(* Schneider Machine Expert - Basic project correto_CORRIGIDO, file version 2.9.0.0 *)
(* ProjectInformations: Name=Novo projeto *)

HARDWARE
  Cpu 0: TM200CE24R
  ModuleExtensionObject 0: TM3TI4/G
  EthernetConfiguration: NetworkName=M200, IpAllocationMode=FixedAddress, IpAddress=192.168.10.1, SubnetMask=255.255.255.0
  SerialLineConfiguration: Baud=Baud9600, Parity=ParityNone, DataBits=DataBits8, StopBits=StopBits1, PhysicalMedium=PhysicalMediumRs485, TransmissionMode=TransmissionModeModbusRtu, SlaveId=1, Addressing=SlaveAddressing
  MastTask: UsePeriodScanMode=true, PeriodScan=10
  FastTask: Period=255
  CpuBehavior: StartingMode=StartAsPreviousState, AutoSaveRamOnEeprom=true, WatchdogPeriod=250

SYMBOLS  (address, symbol, comment, settings)
  %M100     MEM_I00
  %M101     MEM_I01
  %M102     MEM_I02
  %M103     MEM_I03
  %M104     MEM_I04
  %M105     MEM_I05
  %M106     MEM_I06
  %M107     MEM_I07
  %M108     MEM_I08
  %TM0        [Preset=6]
  %TM1        [Preset=2, Base=OneSecond]
  %I0.0     DJ_GERAL_ABERTO
  %I0.1     DJ_GERAL_FECHADO
  %I0.2     RESERVA1
  %I0.3     RESERVA2
  %I0.4     RESERVA3
  %I0.5     RESERVA4
  %I0.6     RESERVA5
  %I0.7     RESERVA6
  %I0.8     RESERVA7
  %I0.9     RESERVA8
  %I0.10    STS_SERVICO_AUX
  %I0.11    BOTAO_CLOSE
  %I0.12    BOTAO_OPEN
  %I0.13    BOTAO_EMERGENCIA
  %Q0.0     COMM_OK
  %Q0.1     USINAGERANDO
  %Q0.2     FALHA
  %Q0.3     ALARME
  %Q0.4     EMERGENCIA_INV
  %Q0.5     RESET_RASP
  %Q0.6     RESET_LINK_3G
  %Q0.7     RESERVA_1
  %Q0.8     RESERVA_2
  %Q0.9     RESERVA_3
  %IW1.0    TEMP_AMBIENTE  [Type=Type_PT100, Scope=Scope_Celsius, Minimum=-2000, Maximum=8500]
  %IW1.1    TEMP_QUADRO  [Type=Type_PT100, Scope=Scope_Celsius, Minimum=-2000, Maximum=8500]
  %IW1.2    TEMP_MODULO  [Type=Type_PT100, Scope=Scope_Celsius, Minimum=-2000, Maximum=8500]
  %IW1.3    TEMP_TRAFO  [Type=Type_PT100, Scope=Scope_Celsius, Minimum=-2000, Maximum=8500]

POU Saídas
  (* SectionNumber=1 *)

// Rung 0: COMUNICAÇÃO OK
  LD %M0
  ST %Q0.0                (* COMM_OK *)
  [ %MW600 := 1 ]
  // as ST:
  //   COMM_OK := %M0;
  //   IF %M0 THEN %MW600 := 1; END_IF;

// Rung 1: STATUS USINA GERANDO
  LD %M1
  ST %Q0.1                (* USINAGERANDO *)
  [ %MW601 := 1 ]
  // as ST:
  //   USINAGERANDO := %M1;
  //   IF %M1 THEN %MW601 := 1; END_IF;

// Rung 2: FALHA
  LD %M2
  ST %Q0.2                (* FALHA *)
  [ %MW602 := 1 ]
  // as ST:
  //   FALHA := %M2;
  //   IF %M2 THEN %MW602 := 1; END_IF;

// Rung 3: ALARME SONORO
  LD %M3
  ST %Q0.3                (* ALARME *)
  [ %MW603 := 1 ]
  // as ST:
  //   ALARME := %M3;
  //   IF %M3 THEN %MW603 := 1; END_IF;

// Rung 4: EMERGÊNCIA INVERSORES
  LDN %I0.13              (* BOTAO_EMERGENCIA *)
  OR %M4
  ST %Q0.4                (* EMERGENCIA_INV *)
  [ %MW604 := 1 ]
  // as ST:
  //   EMERGENCIA_INV := NOT BOTAO_EMERGENCIA OR %M4;
  //   IF NOT BOTAO_EMERGENCIA OR %M4 THEN %MW604 := 1; END_IF;

// Rung 5: RESET LINK 3G
  LD %M6
  ST %Q0.6                (* RESET_LINK_3G *)
  [ %MW606 := 1 ]
  // as ST:
  //   RESET_LINK_3G := %M6;
  //   IF %M6 THEN %MW606 := 1; END_IF;

// Rung 6: RESERVA
  LD %M7
  ST %Q0.7                (* RESERVA_1 *)
  // as ST:
  //   RESERVA_1 := %M7;

// Rung 7: RESERVA
  LD %M8
  ST %Q0.8                (* RESERVA_2 *)
  // as ST:
  //   RESERVA_2 := %M8;

// Rung 8: RESERVA
  LD %M9
  ST %Q0.9                (* RESERVA_3 *)
  // as ST:
  //   RESERVA_3 := %M9;

POU Entradas
  (* SectionNumber=2 *)

// Rung 9: STATUS DISJUNTOR GERAL ABERTO
  LD %I0.0                (* DJ_GERAL_ABERTO *)
  ST %M100                (* MEM_I00 *)
  [ %MW500 := 1 ]
  // as ST:
  //   MEM_I00 := DJ_GERAL_ABERTO;
  //   IF DJ_GERAL_ABERTO THEN %MW500 := 1; END_IF;

// Rung 10: STATUS DISJUNTOR GERAL FECHADO
  LD %I0.1                (* DJ_GERAL_FECHADO *)
  ST %M101                (* MEM_I01 *)
  [ %MW501 := 1 ]
  // as ST:
  //   MEM_I01 := DJ_GERAL_FECHADO;
  //   IF DJ_GERAL_FECHADO THEN %MW501 := 1; END_IF;

// Rung 11: RESERVA
  LD %I0.2                (* RESERVA1 *)
  ST %M102                (* MEM_I02 *)
  // as ST:
  //   MEM_I02 := RESERVA1;

// Rung 12: RESERVA
  LD %I0.3                (* RESERVA2 *)
  ST %M103                (* MEM_I03 *)
  // as ST:
  //   MEM_I03 := RESERVA2;

// Rung 13: RESERVA
  LD %I0.4                (* RESERVA3 *)
  ST %M104                (* MEM_I04 *)
  // as ST:
  //   MEM_I04 := RESERVA3;

// Rung 14: RESERVA
  LD %I0.5                (* RESERVA4 *)
  ST %M105                (* MEM_I05 *)
  // as ST:
  //   MEM_I05 := RESERVA4;

// Rung 15: RESERVA
  LD %I0.6                (* RESERVA5 *)
  ST %M106                (* MEM_I06 *)
  // as ST:
  //   MEM_I06 := RESERVA5;

// Rung 16: RESERVA
  LD %I0.7                (* RESERVA6 *)
  ST %M107                (* MEM_I07 *)
  // as ST:
  //   MEM_I07 := RESERVA6;

// Rung 17: RESERVA
  LD %I0.8                (* RESERVA7 *)
  ST %M108                (* MEM_I08 *)
  // as ST:
  //   MEM_I08 := RESERVA7;

// Rung 18: RESERVA
  LD %I0.9                (* RESERVA8 *)
  ST %M109
  // as ST:
  //   %M109 := RESERVA8;

// Rung 19: STATUS SERVIÇO AUXILIAR
  LD %I0.10               (* STS_SERVICO_AUX *)
  ST %M110
  [ %MW510 := 1 ]
  // as ST:
  //   %M110 := STS_SERVICO_AUX;
  //   IF STS_SERVICO_AUX THEN %MW510 := 1; END_IF;

// Rung 20: BOTÃO FECHA
  LD %I0.11               (* BOTAO_CLOSE *)
  ST %M111
  [ %MW511 := 1 ]
  // as ST:
  //   %M111 := BOTAO_CLOSE;
  //   IF BOTAO_CLOSE THEN %MW511 := 1; END_IF;

// Rung 21: BOTÃO ABRE
  LD %I0.12               (* BOTAO_OPEN *)
  ST %M112
  [ %MW512 := 1 ]
  // as ST:
  //   %M112 := BOTAO_OPEN;
  //   IF BOTAO_OPEN THEN %MW512 := 1; END_IF;

// Rung 22: BOTÃO EMERGÊNCIA
  LDN %I0.13              (* BOTAO_EMERGENCIA *)
  ST %M113
  [ %MW513 := 1 ]
  // as ST:
  //   %M113 := NOT BOTAO_EMERGENCIA;
  //   IF NOT BOTAO_EMERGENCIA THEN %MW513 := 1; END_IF;

POU Analógicas
  (* SectionNumber=3 *)

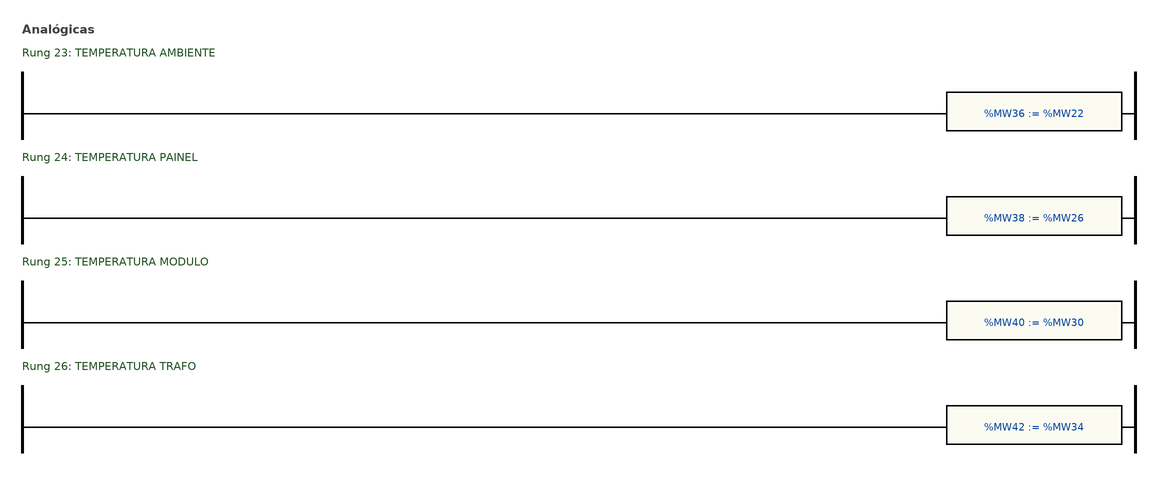

// Rung 23: TEMPERATURA AMBIENTE
  LD 1
  [ %MW36 := %MW22 ]
  // as ST:
  //   %MW36 := %MW22;

// Rung 24: TEMPERATURA PAINEL
  LD 1
  [ %MW38 := %MW26 ]
  // as ST:
  //   %MW38 := %MW26;

// Rung 25: TEMPERATURA MODULO
  LD 1
  [ %MW40 := %MW30 ]
  // as ST:
  //   %MW40 := %MW30;

// Rung 26: TEMPERATURA TRAFO
  LD 1
  [ %MW42 := %MW34 ]
  // as ST:
  //   %MW42 := %MW34;

POU ESCALA TEMPERATURA
  (* SectionNumber=4 *)

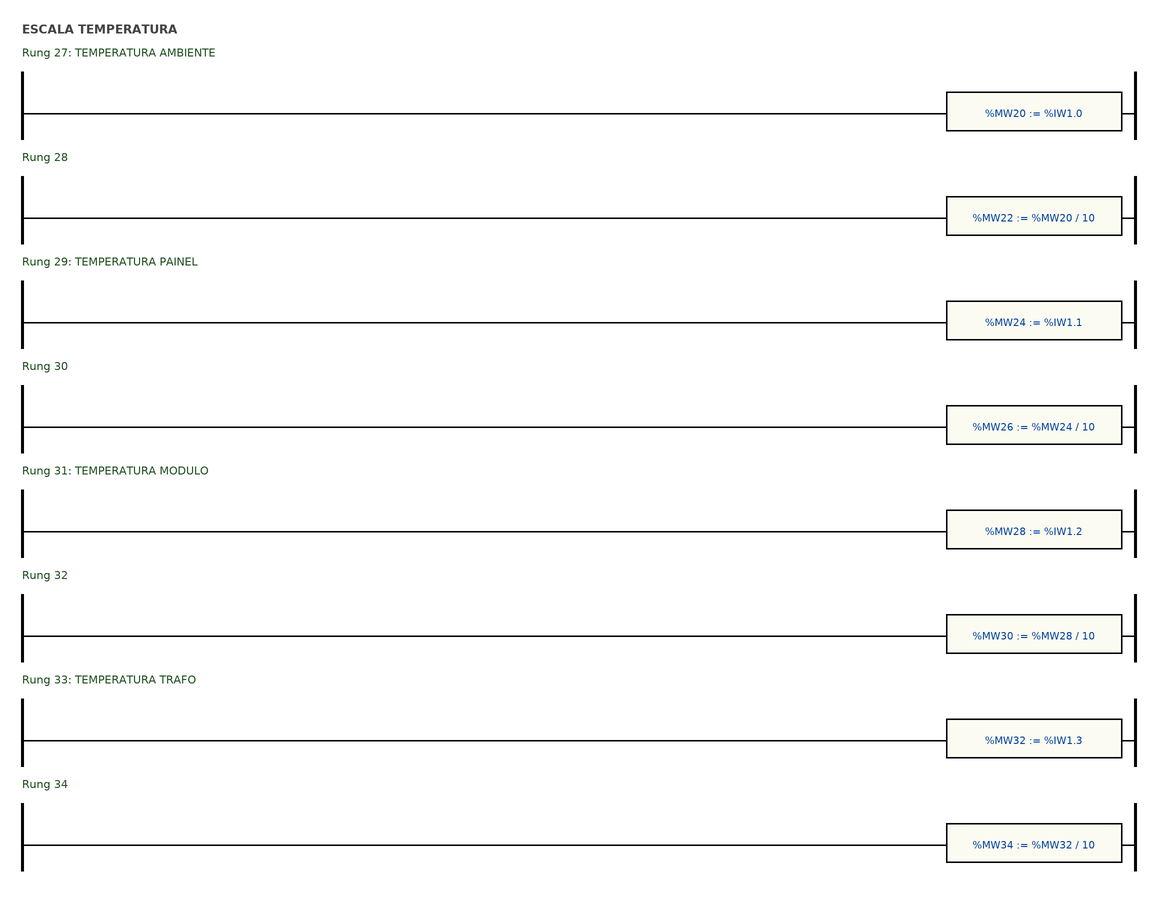

// Rung 27: TEMPERATURA AMBIENTE
  LD 1
  [ %MW20 := %IW1.0 ]     (* TEMP_AMBIENTE *)
  // as ST:
  //   %MW20 := TEMP_AMBIENTE;

// Rung 28
  LD 1
  [ %MW22 := %MW20 / 10 ]
  // as ST:
  //   %MW22 := %MW20 / 10;

// Rung 29: TEMPERATURA PAINEL
  LD 1
  [ %MW24 := %IW1.1 ]     (* TEMP_QUADRO *)
  // as ST:
  //   %MW24 := TEMP_QUADRO;

// Rung 30
  LD 1
  [ %MW26 := %MW24 / 10 ]
  // as ST:
  //   %MW26 := %MW24 / 10;

// Rung 31: TEMPERATURA MODULO
  LD 1
  [ %MW28 := %IW1.2 ]     (* TEMP_MODULO *)
  // as ST:
  //   %MW28 := TEMP_MODULO;

// Rung 32
  LD 1
  [ %MW30 := %MW28 / 10 ]
  // as ST:
  //   %MW30 := %MW28 / 10;

// Rung 33: TEMPERATURA TRAFO
  LD 1
  [ %MW32 := %IW1.3 ]     (* TEMP_TRAFO *)
  // as ST:
  //   %MW32 := TEMP_TRAFO;

// Rung 34
  LD 1
  [ %MW34 := %MW32 / 10 ]
  // as ST:
  //   %MW34 := %MW32 / 10;

POU Reset Raspberry
  (* SectionNumber=5 *)

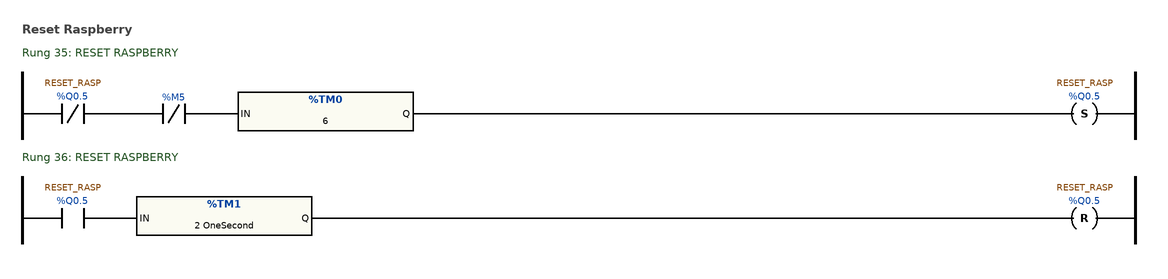

// Rung 35: RESET RASPBERRY
  BLK %TM0
  LDN %Q0.5               (* RESET_RASP *)
  ANDN %M5
  IN
  OUT_BLK
  LD Q
  S %Q0.5                 (* RESET_RASP *)
  END_BLK
  // as ST:
  //   %TM0(IN := NOT RESET_RASP AND NOT %M5);
  //   IF %TM0.Q THEN RESET_RASP := TRUE; END_IF;

// Rung 36: RESET RASPBERRY
  BLK %TM1
  LD %Q0.5                (* RESET_RASP *)
  IN
  OUT_BLK
  LD Q
  R %Q0.5                 (* RESET_RASP *)
  END_BLK
  // as ST:
  //   %TM1(IN := RESET_RASP);
  //   IF %TM1.Q THEN RESET_RASP := FALSE; END_IF;

POU Mapeamento Modbus
  (* SectionNumber=6 *)

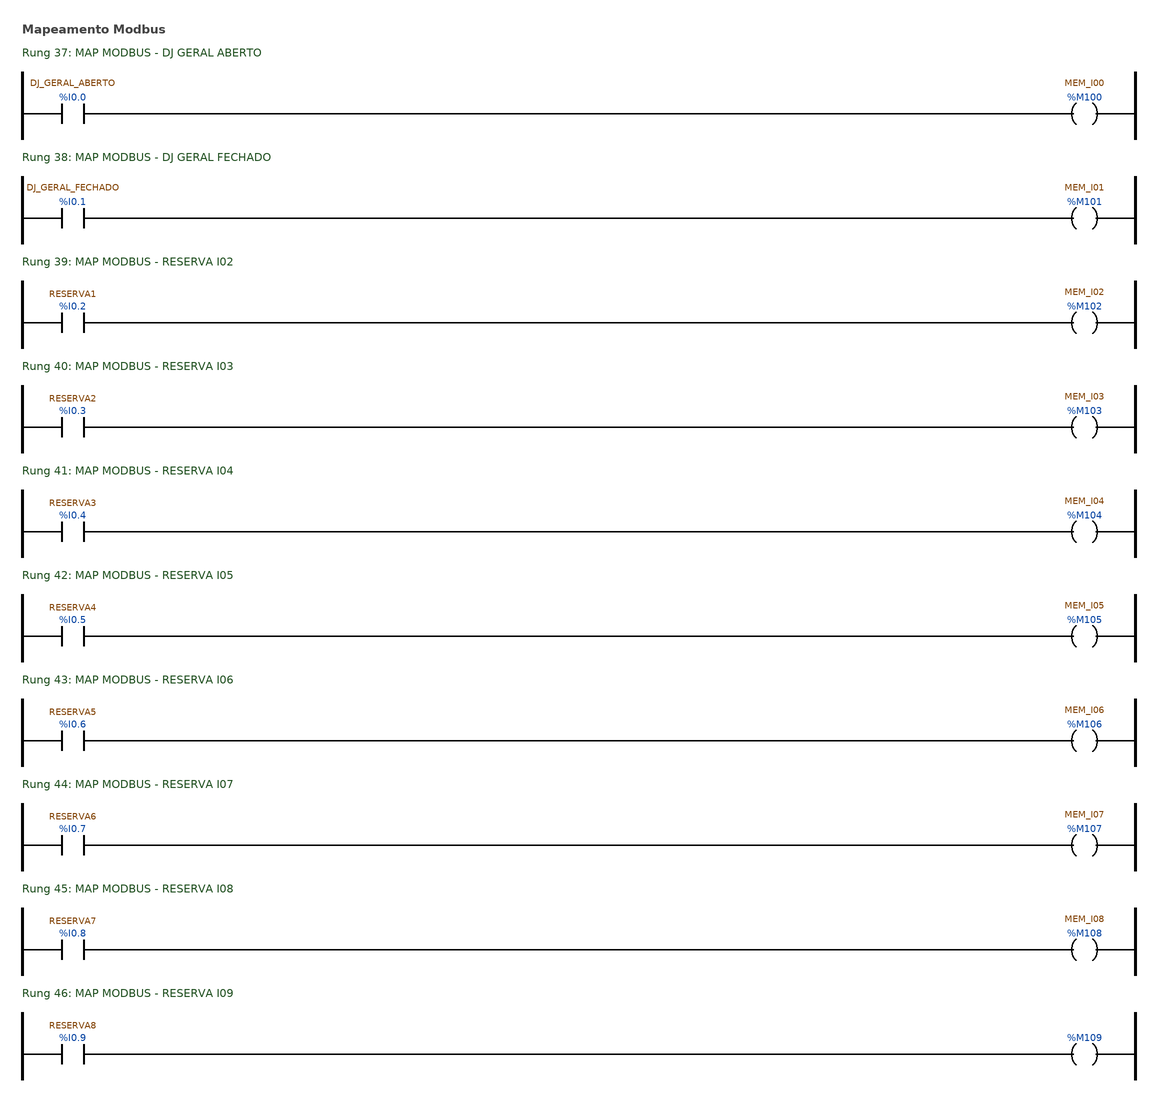

// Rung 37: MAP MODBUS - DJ GERAL ABERTO
  LD %I0.0                (* DJ_GERAL_ABERTO *)
  ST %M100                (* MEM_I00 *)
  // as ST:
  //   MEM_I00 := DJ_GERAL_ABERTO;

// Rung 38: MAP MODBUS - DJ GERAL FECHADO
  LD %I0.1                (* DJ_GERAL_FECHADO *)
  ST %M101                (* MEM_I01 *)
  // as ST:
  //   MEM_I01 := DJ_GERAL_FECHADO;

// Rung 39: MAP MODBUS - RESERVA I02
  LD %I0.2                (* RESERVA1 *)
  ST %M102                (* MEM_I02 *)
  // as ST:
  //   MEM_I02 := RESERVA1;

// Rung 40: MAP MODBUS - RESERVA I03
  LD %I0.3                (* RESERVA2 *)
  ST %M103                (* MEM_I03 *)
  // as ST:
  //   MEM_I03 := RESERVA2;

// Rung 41: MAP MODBUS - RESERVA I04
  LD %I0.4                (* RESERVA3 *)
  ST %M104                (* MEM_I04 *)
  // as ST:
  //   MEM_I04 := RESERVA3;

// Rung 42: MAP MODBUS - RESERVA I05
  LD %I0.5                (* RESERVA4 *)
  ST %M105                (* MEM_I05 *)
  // as ST:
  //   MEM_I05 := RESERVA4;

// Rung 43: MAP MODBUS - RESERVA I06
  LD %I0.6                (* RESERVA5 *)
  ST %M106                (* MEM_I06 *)
  // as ST:
  //   MEM_I06 := RESERVA5;

// Rung 44: MAP MODBUS - RESERVA I07
  LD %I0.7                (* RESERVA6 *)
  ST %M107                (* MEM_I07 *)
  // as ST:
  //   MEM_I07 := RESERVA6;

// Rung 45: MAP MODBUS - RESERVA I08
  LD %I0.8                (* RESERVA7 *)
  ST %M108                (* MEM_I08 *)
  // as ST:
  //   MEM_I08 := RESERVA7;

// Rung 46: MAP MODBUS - RESERVA I09
  LD %I0.9                (* RESERVA8 *)
  ST %M109
  // as ST:
  //   %M109 := RESERVA8;

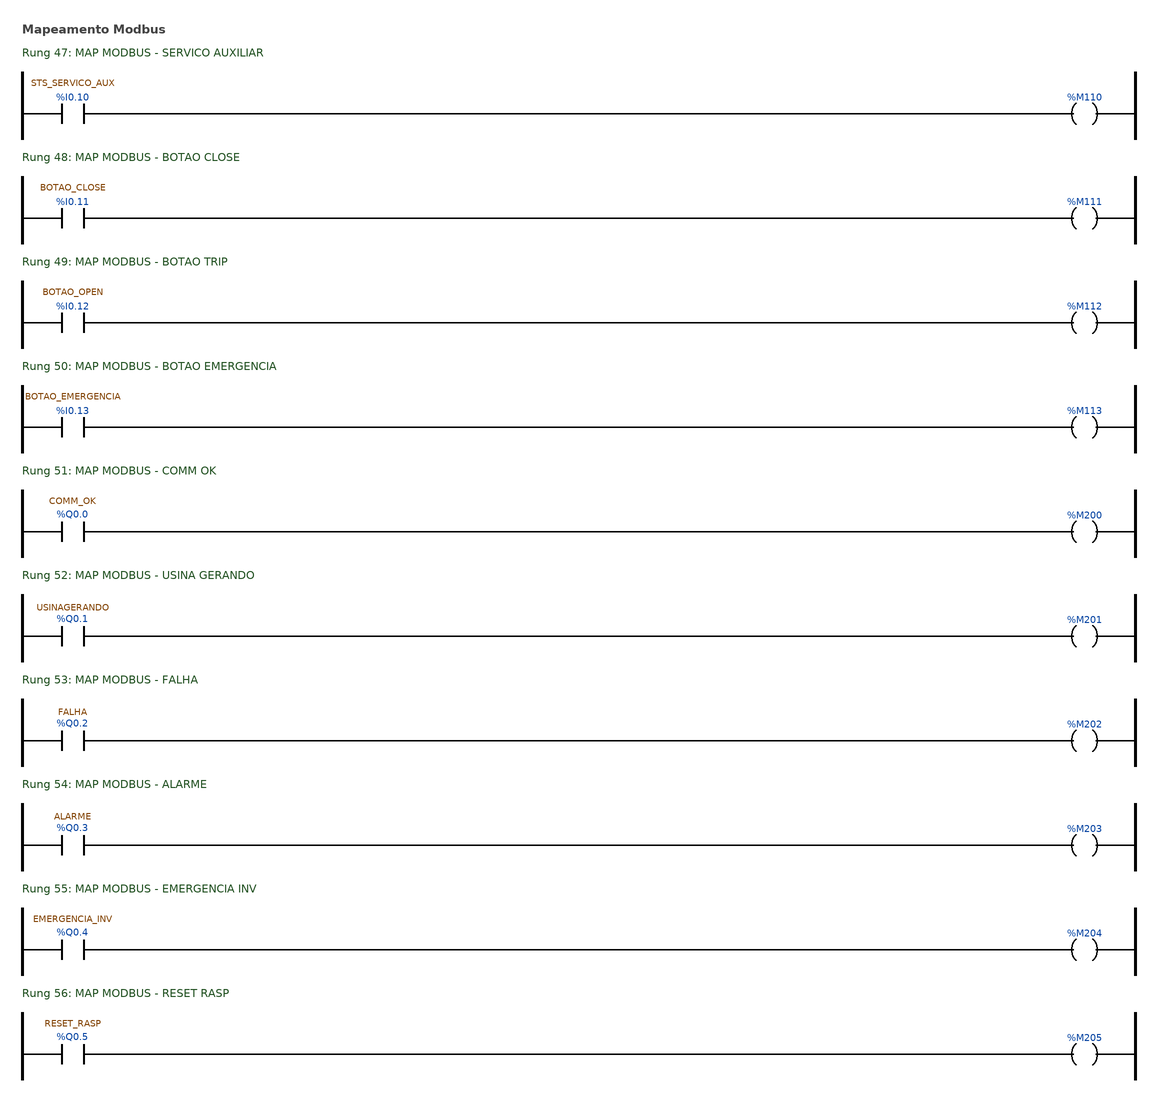

// Rung 47: MAP MODBUS - SERVICO AUXILIAR
  LD %I0.10               (* STS_SERVICO_AUX *)
  ST %M110
  // as ST:
  //   %M110 := STS_SERVICO_AUX;

// Rung 48: MAP MODBUS - BOTAO CLOSE
  LD %I0.11               (* BOTAO_CLOSE *)
  ST %M111
  // as ST:
  //   %M111 := BOTAO_CLOSE;

// Rung 49: MAP MODBUS - BOTAO TRIP
  LD %I0.12               (* BOTAO_OPEN *)
  ST %M112
  // as ST:
  //   %M112 := BOTAO_OPEN;

// Rung 50: MAP MODBUS - BOTAO EMERGENCIA
  LD %I0.13               (* BOTAO_EMERGENCIA *)
  ST %M113
  // as ST:
  //   %M113 := BOTAO_EMERGENCIA;

// Rung 51: MAP MODBUS - COMM OK
  LD %Q0.0                (* COMM_OK *)
  ST %M200
  // as ST:
  //   %M200 := COMM_OK;

// Rung 52: MAP MODBUS - USINA GERANDO
  LD %Q0.1                (* USINAGERANDO *)
  ST %M201
  // as ST:
  //   %M201 := USINAGERANDO;

// Rung 53: MAP MODBUS - FALHA
  LD %Q0.2                (* FALHA *)
  ST %M202
  // as ST:
  //   %M202 := FALHA;

// Rung 54: MAP MODBUS - ALARME
  LD %Q0.3                (* ALARME *)
  ST %M203
  // as ST:
  //   %M203 := ALARME;

// Rung 55: MAP MODBUS - EMERGENCIA INV
  LD %Q0.4                (* EMERGENCIA_INV *)
  ST %M204
  // as ST:
  //   %M204 := EMERGENCIA_INV;

// Rung 56: MAP MODBUS - RESET RASP
  LD %Q0.5                (* RESET_RASP *)
  ST %M205
  // as ST:
  //   %M205 := RESET_RASP;

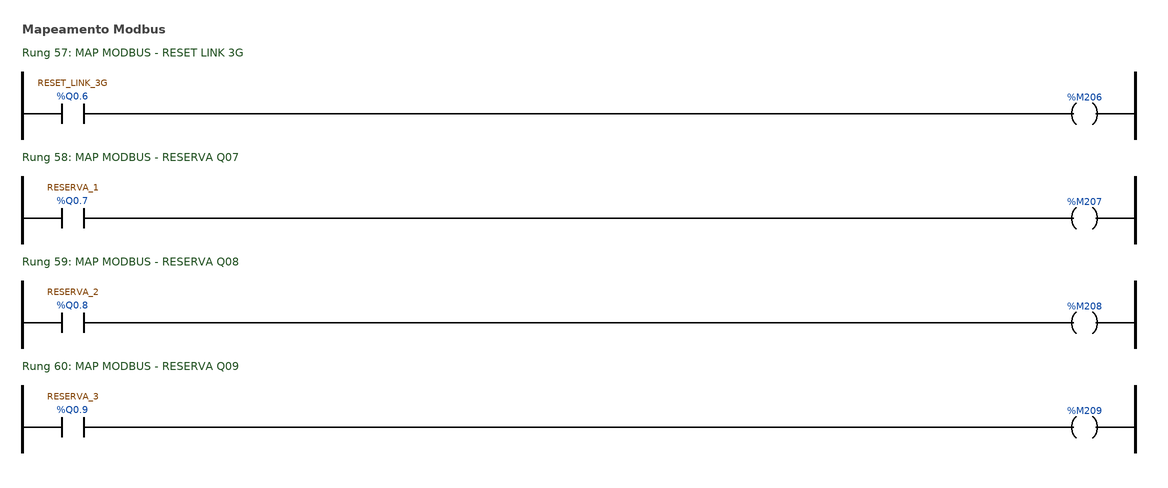

// Rung 57: MAP MODBUS - RESET LINK 3G
  LD %Q0.6                (* RESET_LINK_3G *)
  ST %M206
  // as ST:
  //   %M206 := RESET_LINK_3G;

// Rung 58: MAP MODBUS - RESERVA Q07
  LD %Q0.7                (* RESERVA_1 *)
  ST %M207
  // as ST:
  //   %M207 := RESERVA_1;

// Rung 59: MAP MODBUS - RESERVA Q08
  LD %Q0.8                (* RESERVA_2 *)
  ST %M208
  // as ST:
  //   %M208 := RESERVA_2;

// Rung 60: MAP MODBUS - RESERVA Q09
  LD %Q0.9                (* RESERVA_3 *)
  ST %M209
  // as ST:
  //   %M209 := RESERVA_3;
